FUNCTION_BLOCK FB_Communication
VAR_INPUT
END_VAR
VAR_OUTPUT
END_VAR

VAR_IN_OUT
	stAxisStruct			: AxisStruct;
END_VAR

VAR
	bStart					: BOOL;
	bError					: BOOL;
	nErrorID				: LREAL;
	bStop					: BOOL;
	bReset					: BOOL;
	bResetDone				: BOOL;
	bEnabled				: BOOL;
	eCommState				: CommStates;
	bFirstScan				: BOOL:= TRUE;
	fbRTrig_StartMov		: R_trig;
	
END_VAR

fbRTrig_StartMov(CLK:= stAxisStruct.bStart AND eCommState = 1);
//bStart	:= stAxisStruct.bStart;
//bStop	:= stAxisStruct.bStop;
//bReset	:= stAxisStruct.bReset;
//bResetDone := stAxisStruct.bResetDone;
//bEnabled	:= stAxisStruct.bEnabled; come from FB_DriveVirtual
stAxisStruct.Axis.ReadStatus();
IF NOT stAxisStruct.bEnabled AND stAxisStruct.Axis.Status.Disabled THEN 
	eCommState := 2; //disabled
ELSIF NOT stAxisStruct.bReset AND  stAxisStruct.Axis.Status.Error THEN 
	eCommState := 8; //ERROR
ELSIF stAxisStruct.bReset THEN
	eCommState := 0;
END_IF

CASE eCommState OF
        0 : (* Reset (error-ACK) *)
			IF stAxisStruct.bError AND NOT stAxisStruct.bResetDone THEN 
					eCommState := 0; //Reset not finished
			ELSIF stAxisStruct.Axis.Status.StandStill AND NOT stAxisStruct.bReset THEN //reset done jump to idle
					eCommState := 1;
			END_IF
						
		2: (*Enable, disabled*)
			IF stAxisStruct.bEnabled AND NOT stAxisStruct.bError THEN
				eCommState := 1;
			ELSIF stAxisStruct.bError THEN
				eCommState := 8;
			ELSE
				eCommState := 2;
			END_IF
		1,3: (* idle, warn *)
             (* XXX: check enable? limit switches? *)
			IF stAxisStruct.bStop THEN
				eCommState := 7;
			ELSIF fbRTrig_StartMov.Q THEN
				eCommState:= 5;
			ELSIF stAxisStruct.Axis.Status.Moving THEN
				eCommState:= 6;
			ELSE
				eCommState:= 1;
			END_IF
			//bJogBwd := bStartJogBwd;
			//bJogFwd := bStartJogFwd;
			//bHome;
           
		5:  (* START *)
			IF stAxisStruct.Axis.Status.HasJob THEN
				eCommState := 6;
			ELSIF stAxisStruct.Axis.Status.StandStill THEN
				eCommState := 1;		
			END_IF
		    //add a Ontaget siganl or use bDone?????
        6:  (* BUSY *)
			IF stAxisStruct.Axis.Status.Stopping THEN 
				eCommState := 7;
			ELSIF stAxisStruct.Axis.Status.StandStill AND NOT stAxisStruct.Axis.Status.HasJob THEN
				eCommState := 1;
          	END_IF
			
		7:  (* STOP *)
			IF stAxisStruct.Axis.Status.Stopping THEN
				eCommState := 7;
			ELSIF stAxisStruct.Axis.Status.StandStill THEN
				eCommState := 1;
			END_IF
  
        8:  (* ERROR *)
			stAxisStruct.bError := TRUE;
			stAxisStruct.nErrorID := stAxisStruct.Axis.Status.ErrorID;
			IF stAxisStruct.bReset THEN
				eCommState := 0;
			END_IF
            
    END_CASE

IF bFirstScan THEN
	bFirstScan:=FALSE;
END_IF

END_FUNCTION_BLOCK

(* stored: Version 1.1.0.1, ProductVersion 3.1.4022.17
   POU FB_Communication: Id {71515715-1dbd-4921-bede-91a04a907ca4}, SpecialFunc None *)
